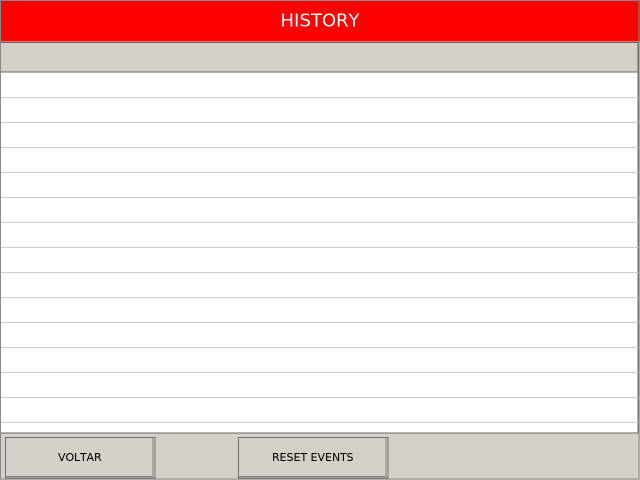
VISUALIZATION VISU_EVENTS  // 640x480
    Button (5,437 150x41), "VOLTAR"
        OnMouseClick: change screen: VISU_MAIN
    Table (0,42 638x391), data array: GVL_ALARMS.HISTORY_ALARMS
        p3854506369: GVL_ALARMS.HISTORY_ALARMS[INDEX].byGroup
        p1892666644: GVL_ALARMS.HISTORY_ALARMS[INDEX].sDate_on
        p338671338: GVL_ALARMS.HISTORY_ALARMS[INDEX].sHour_on
        p2170511999: GVL_ALARMS.HISTORY_ALARMS[INDEX].sDate_off
        p3723444502: GVL_ALARMS.HISTORY_ALARMS[INDEX].sHour_off
        p1218418051: GVL_ALARMS.HISTORY_ALARMS[INDEX].iNumber
        p746581629: GVL_ALARMS.HISTORY_ALARMS[INDEX].dwTextColor
        p511219082: DATA IN
        p1755163831: HORA IN
        p4092479075: DATA OFF
        p2237128397: HORA OFF
    Rectangle (0,0 640x41), "HISTORY"
    Button (238,437 150x41), "RESET EVENTS"
        tap GVL_ALARMS.bResetEvents
END_VISUALIZATION

(* stored: Version 1.1.0.1, ProductVersion 3.1.4024.12
   Visu VISU_EVENTS: Id {b10aa941-5d87-41d6-84f6-ffe062725151} *)
